TYPE E_BCD_Type :
(
	None := 0,
	SICK,
	KEYENCE
);
END_TYPE

(* stored: Version 1.1.0.1, ProductVersion 3.1.0.26
   DUT E_BCD_Type: Id {2c07d06e-e910-44fe-a4e8-69b111a759ce} *)
